FUNCTION_BLOCK Sensor_Comunicacao (* Composite Function Block Type *)
  (* Standard: 61499-2 *)
  (* Version 0.0, 20/01/2026, Schneider Electric, template *)
  PACKAGE Hidryco.HidrycoLib;
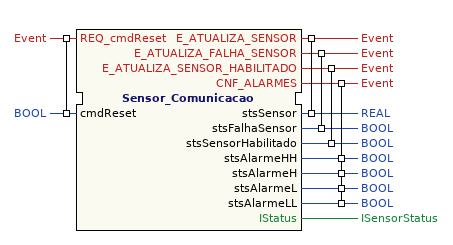
  EVENT_INPUT
    REQ_cmdReset WITH cmdReset;
  END_EVENT
  EVENT_OUTPUT
    E_ATUALIZA_SENSOR WITH stsSensor;
    E_ATUALIZA_FALHA_SENSOR WITH stsFalhaSensor;
    E_ATUALIZA_SENSOR_HABILITADO WITH stsSensorHabilitado;
    CNF_ALARMES WITH stsAlarmeHH, stsAlarmeH, stsAlarmeL, stsAlarmeLL;
  END_EVENT
  VAR_INPUT
    cmdReset : BOOL;
  END_VAR
  VAR_OUTPUT
    stsSensor : REAL;
    stsFalhaSensor : BOOL;
    stsSensorHabilitado : BOOL;
    stsAlarmeHH : BOOL; (* Output event qualifier *)
    stsAlarmeH : BOOL;
    stsAlarmeL : BOOL;
    stsAlarmeLL : BOOL;
  END_VAR
  PLUGS
    IStatus : ISensorStatus;
  END_PLUGS
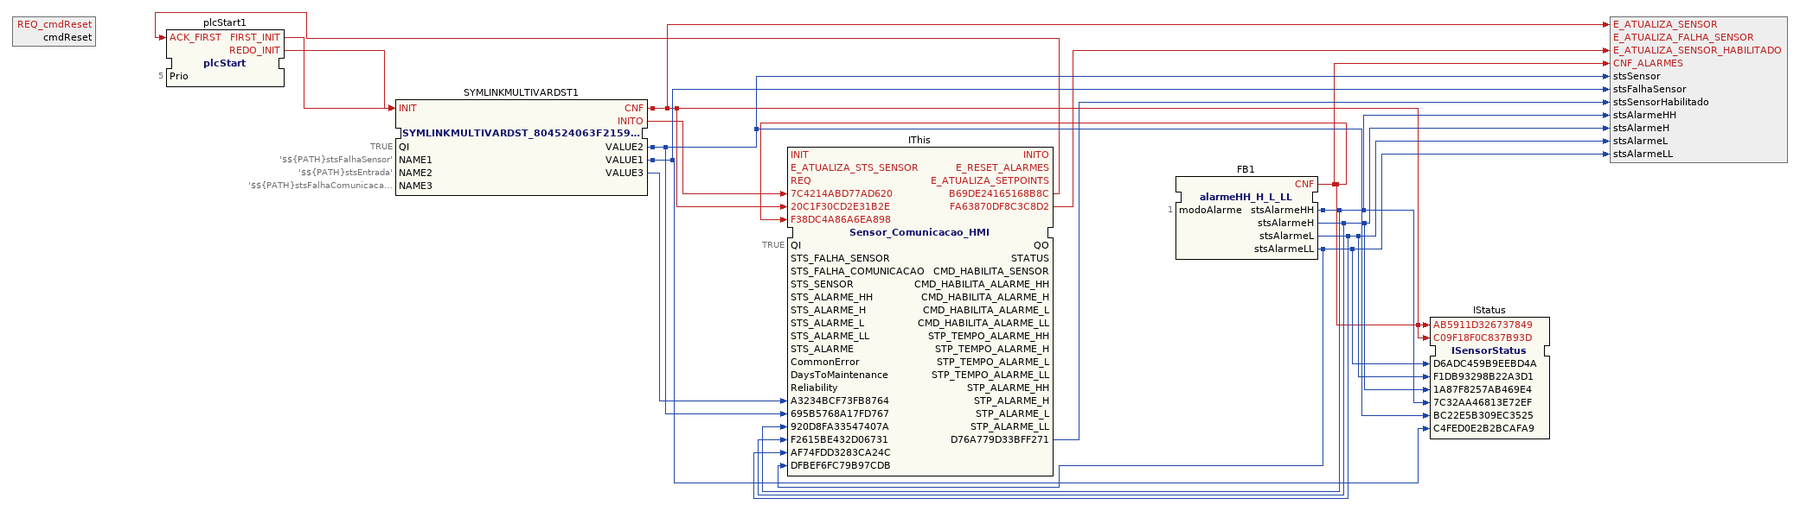
  FBS
    FB1 : alarmeHH_H_L_LL(modoAlarme := 1);
    IThis : Sensor_Comunicacao_HMI(QI := TRUE);
    SYMLINKMULTIVARDST1 : SYMLINKMULTIVARDST_804524063F215924(QI := TRUE, NAME1 := '$${PATH}stsFalhaSensor', NAME2 := '$${PATH}stsEntrada', NAME3 := '$${PATH}stsFalhaComunicacao'); {SET_ATTRIBUTE(Configuration.GenericFBType.InterfaceParams, Runtime.System#I:=3;VALUE${I$}:BOOL,REAL,BOOL)}
    plcStart1 : plcStart(Prio := 5);
  END_FBS
  EVENT_CONNECTIONS
    FB1.CNF TO CNF_ALARMES;
    FB1.CNF TO IStatus.AB5911D326737849;
    plcStart1.FIRST_INIT TO SYMLINKMULTIVARDST1.INIT;
    plcStart1.REDO_INIT TO SYMLINKMULTIVARDST1.INIT;
    SYMLINKMULTIVARDST1.CNF TO E_ATUALIZA_SENSOR;
    SYMLINKMULTIVARDST1.CNF TO IStatus.C09F18F0C837B93D;
    SYMLINKMULTIVARDST1.INITO TO IThis.7C4214ABD77AD620;
    SYMLINKMULTIVARDST1.CNF TO IThis.20C1F30CD2E31B2E;
    FB1.CNF TO IThis.F38DC4A86A6EA898;
    IThis.B69DE24165168B8C TO plcStart1.ACK_FIRST;
    IThis.FA63870DF8C3C8D2 TO E_ATUALIZA_SENSOR_HABILITADO;
    SYMLINKMULTIVARDST1.CNF TO IStatus.AB5911D326737849;
  END_CONNECTIONS
  DATA_CONNECTIONS
    FB1.stsAlarmeHH TO stsAlarmeHH;
    FB1.stsAlarmeH TO stsAlarmeH;
    FB1.stsAlarmeL TO stsAlarmeL;
    FB1.stsAlarmeLL TO stsAlarmeLL;
    FB1.stsAlarmeLL TO IStatus.D6ADC459B9EEBD4A;
    FB1.stsAlarmeL TO IStatus.F1DB93298B22A3D1;
    FB1.stsAlarmeH TO IStatus.1A87F8257AB469E4;
    FB1.stsAlarmeHH TO IStatus.7C32AA46813E72EF;
    SYMLINKMULTIVARDST1.VALUE2 TO stsSensor;
    SYMLINKMULTIVARDST1.VALUE2 TO IStatus.BC22E5B309EC3525;
    SYMLINKMULTIVARDST1.VALUE1 TO stsFalhaSensor;
    SYMLINKMULTIVARDST1.VALUE1 TO IStatus.C4FED0E2B2BCAFA9;
    SYMLINKMULTIVARDST1.VALUE3 TO IThis.A3234BCF73FB8764;
    SYMLINKMULTIVARDST1.VALUE2 TO IThis.695B5768A17FD767;
    FB1.stsAlarmeHH TO IThis.920D8FA33547407A;
    FB1.stsAlarmeH TO IThis.F2615BE432D06731;
    FB1.stsAlarmeL TO IThis.AF74FDD3283CA24C;
    FB1.stsAlarmeLL TO IThis.DFBEF6FC79B97CDB;
    IThis.D76A779D33BFF271 TO stsSensorHabilitado;
  END_CONNECTIONS
END_FUNCTION_BLOCK
